FUNCTION_BLOCK fail_scenarios1 (* Composite Function Block Type *)
  (* Standard: 61499-2 *)
  (* Version 0.0, 5/15/2019, erik, nxtControl GmbH, template *)
  PACKAGE Main;
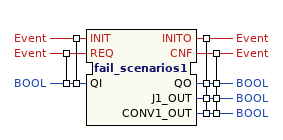
  EVENT_INPUT
    INIT WITH QI; (* Initialization Request *)
    REQ WITH QI; (* Normal Execution Request *)
  END_EVENT
  EVENT_OUTPUT
    INITO WITH QO, J1_OUT, CONV1_OUT; (* Initialization Confirm *)
    CNF WITH QO, J1_OUT, CONV1_OUT; (* Execution Confirmation *)
  END_EVENT
  VAR_INPUT
    QI : BOOL; (* Input event qualifier *)
  END_VAR
  VAR_OUTPUT
    QO : BOOL; (* Output event qualifier *)
    J1_OUT : BOOL := TRUE;
    CONV1_OUT : BOOL := TRUE;
  END_VAR
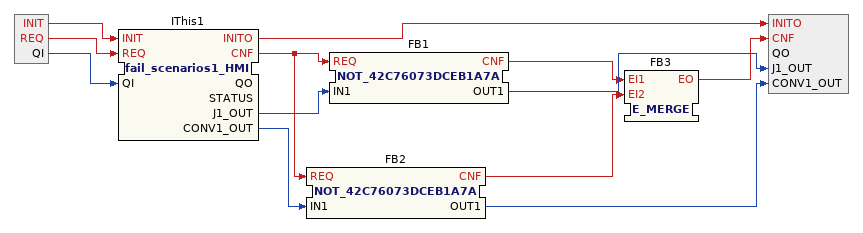
  FBS
    IThis1 : fail_scenarios1_HMI;
    FB1 : NOT_42C76073DCEB1A7A; {SET_ATTRIBUTE(Configuration.GenericFBType.InterfaceParams, Runtime.Standard#CNT:=1;OUT${CNT$}:BOOL)}
    FB2 : NOT_42C76073DCEB1A7A; {SET_ATTRIBUTE(Configuration.GenericFBType.InterfaceParams, Runtime.Standard#CNT:=1;OUT${CNT$}:BOOL)}
    FB3 : E_MERGE;
  END_FBS
  EVENT_CONNECTIONS
    INIT TO IThis1.INIT;
    REQ TO IThis1.REQ;
    IThis1.INITO TO INITO;
    IThis1.CNF TO FB1.REQ;
    IThis1.CNF TO FB2.REQ;
    FB3.EO TO CNF;
    FB1.CNF TO FB3.EI1;
    FB2.CNF TO FB3.EI2;
  END_CONNECTIONS
  DATA_CONNECTIONS
    FB1.OUT1 TO J1_OUT;
    FB2.OUT1 TO CONV1_OUT;
    QI TO IThis1.QI;
    IThis1.J1_OUT TO FB1.IN1;
    IThis1.CONV1_OUT TO FB2.IN1;
  END_CONNECTIONS
END_FUNCTION_BLOCK
